PROGRAM POU
VAR
	T1: TON;
	TON_0:TON;
    Cycle: BOOL;
END_VAR
VAR // added by the converter: edge detectors and wires of the graphical bodies
    _w1 : BOOL;
END_VAR

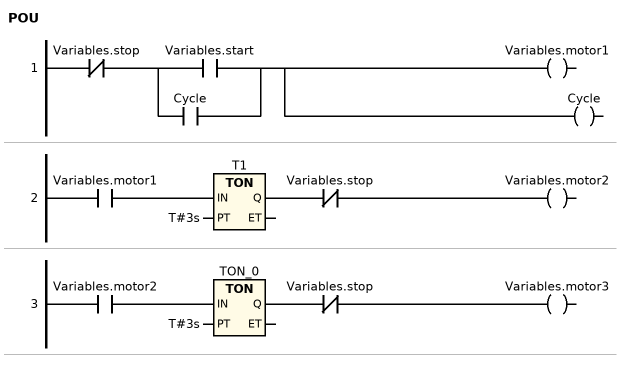
// NETWORK 1
_w1 := NOT Variables.stop AND (Variables.start OR Cycle);
Variables.motor1 := _w1;
Cycle := _w1;

// NETWORK 2
T1(IN := Variables.motor1, PT := T#3s); // TON
Variables.motor2 := T1.Q AND NOT Variables.stop;

// NETWORK 3
TON_0(IN := Variables.motor2, PT := T#3s); // TON
Variables.motor3 := TON_0.Q AND NOT Variables.stop;

END_PROGRAM

(* stored: Version 1.1.0.1, ProductVersion 3.1.4024.12
   POU POU: Id {a9466a27-dd51-4e58-abeb-ec06a7aafb4b}, SpecialFunc None *)
